TYPE DUT_HMI_05_MANUALS :
STRUCT
	PS : ARRAY[0..CNC.NUM_MAX_MANUALS_05-1] OF BOOL;
	LS : ARRAY[0..CNC.NUM_MAX_MANUALS_05-1] OF BOOL;
END_STRUCT
END_TYPE

(* stored: Version 1.1.0.1, ProductVersion 3.1.4024.13
   DUT DUT_HMI_05_MANUALS: Id {782449e0-c9c8-4252-a444-e9eed52cc42b} *)
